// Attempts to dereference a pointer up to a given number of levels.
// [note] the given pointer is returned if Levels is 0.
FUNCTION F_TryDerefPointer : POINTER TO BYTE // Final dereferenced pointer or 0 if not readable.
VAR_INPUT
	// Pointer to start dereferencing from.
	pValue : POINTER TO BYTE;
	// Number of dereference levels to attempt.
	Levels : T_Size;
END_VAR
VAR
	i 		: T_Position;
	pTmp 	: POINTER TO POINTER TO BYTE;
END_VAR

// Return the same pointer of 0 levels.
pTmp := F_TryDerefPointer := pValue;

FOR i := 1 TO Levels DO
	RETURN(NOT F_IsReadablePointer(F_TryDerefPointer));
	pTmp := F_TryDerefPointer;
	F_TryDerefPointer := pTmp^;
	END_FOR

END_FUNCTION

(* stored: Version 1.1.0.1
   POU F_TryDerefPointer: Id {db7a4388-c12a-05b8-3a80-c5e1220360cd}, SpecialFunc None *)
